PROGRAM P_Task2
VAR
END_VAR

END_PROGRAM

(* stored: Version 1.1.0.1, ProductVersion 3.1.4024.12
   POU P_Task2: Id {a6b437aa-74eb-4ef9-8a51-13b0b8f805bf}, SpecialFunc None *)
